FUNCTION_BLOCK Toggle (* Basic Function Block Type *)
  (* Standard: 61499-2 *)
  (* Version 0.0, 10/14/2015, embsys, nxtControl GmbH, Template *)
  PACKAGE Main;
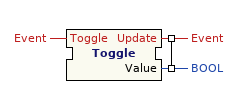
  EVENT_INPUT
    Toggle; (* Normal Execution Request *)
  END_EVENT
  EVENT_OUTPUT
    Update WITH Value; (* Execution Confirmation *)
  END_EVENT
  VAR_OUTPUT
    Value : BOOL; (* Output event qualifier *)
  END_VAR
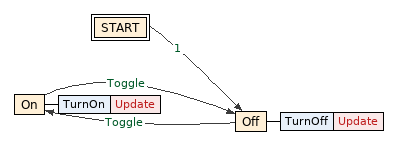
  EC_STATES
    START; (* Initial State *)
    On : TurnOn -> Update; (* Normal execution *)
    Off : TurnOff -> Update;
  END_STATES
  EC_TRANSITIONS
    START TO Off := 1;
    Off TO On := Toggle;
    On TO Off := Toggle;
  END_TRANSITIONS
  ALGORITHM TurnOn IN ST: (* Normally executed algorithm *)
Value:=TRUE;
  END_ALGORITHM
  ALGORITHM TurnOff IN ST:
Value:=FALSE;
  END_ALGORITHM
END_FUNCTION_BLOCK
